TYPE ST_RGB :
STRUCT
	red		:	BYTE;
	green	:	BYTE;
	blue	:	BYTE;
END_STRUCT
END_TYPE

(* stored: Version 1.1.0.1, ProductVersion 3.1.4024.12
   DUT ST_RGB: Id {78bb5374-addf-4e76-a7c4-de48a3eeccde} *)
